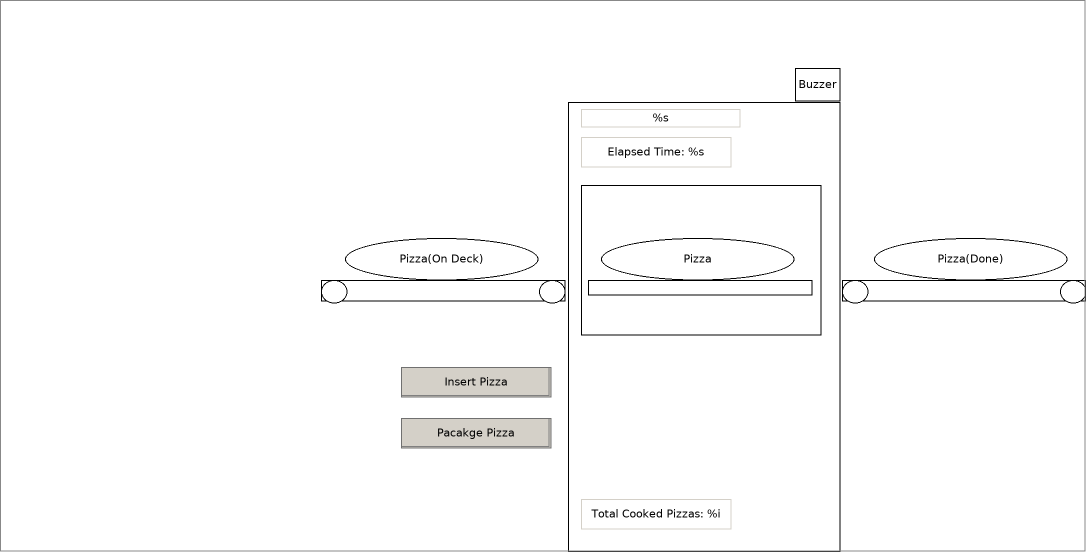
VISUALIZATION Visualization  // 1086x552
    Rectangle (568,102 272x450)
    Button (401,367 150x30), "Insert Pizza", pressed state: MAIN.bPizzaOnDeck
        OnMouseClick: execute { MAIN.bPizzaInOven := TRUE ; }
    Button (401,418 150x30), "Pacakge Pizza"
        OnMouseClick: execute { MAIN.bPizzaInOven := FALSE }
    Rectangle (581,185 240x150)
    Ellipse (601,238 193x42), "Pizza", invisible if: NOT MAIN.bPizzaInOven
    Textfield (581,137 150x30), "Elapsed Time: %s", text variable: MAIN.fbTimer.ET
    Textfield (581,499 150x30), "Total Cooked Pizzas: %i", text variable: MAIN.nTotalPizzasCooked
    Rectangle (321,280 244x21)
    Ellipse (321,280 26x23)
    Ellipse (539,280 26x23)
    Rectangle (588,280 224x15)
    Rectangle (842,280 244x21)
    Ellipse (842,280 26x23)
    Ellipse (1060,280 26x23)
    Ellipse (345,238 193x42), "Pizza(On Deck)", invisible if: NOT MAIN.bPizzaOnDeck
    Ellipse (874,238 193x42), "Pizza(Done)", invisible if: NOT MAIN.bPizzaDone
    Rectangle (795,68 45x33), "Buzzer", colour toggle: MAIN.bBuzzer
    Textfield (581,109 159x18), "%s", text variable: MAIN.sCurrentStateString
END_VISUALIZATION

(* stored: Version 1.1.0.1
   Visu Visualization: Id {98b3cb9e-bb5a-41e0-ae95-282ced915911} *)
